// TIA Portal V17 export
// export: Created 2022-07-20T07:02:40.1160452Z, ExportSetting WithDefaults, DisplayName Totally Integrated Automation Portal, DisplayVersion V17, DisplayName TIA Portal Openness, DisplayVersion V17, DisplayName TIA Portal Version Control Interface, DisplayVersion V17, DisplayName SINAMICS Startdrive Advanced, DisplayVersion V17, DisplayName SINAMICS Startdrive G130, G150, S120, S150, SINAMICS MV, S210, DisplayVersion V17, DisplayName SINAMICS Startdrive G110M, G120, G120C, G120D, G120P, G115D, DisplayVersion V17, DisplayName STEP 7 Professional, DisplayVersion V17, DisplayName STEP 7 Safety, DisplayVersion V17, DisplayName WinCC Advanced, DisplayVersion V17
VAR_GLOBAL   // PLC tag table "LAcycCom_Drives"
END_VAR
VAR_GLOBAL CONSTANT   // user constants
   LACYCCOM_WRITE_PARAMETERS_UPPER_LIM : Int := 18;
   LACYCCOM_READ_PARAMETERS_UPPER_LIM : Int := 38;
   LACYCCOM_SILENT_OPERATION_PARAMETERS_UPPER_LIM : Int := 17;
   LACYCCOM_NO_COMMAND : Byte := 16#00;
   LACYCCOM_READ_COMMAND : Byte := 16#01;
   LACYCCOM_WRITE_COMMAND : Byte := 16#02;
   LACYCCOM_TYPE_ALARM : SInt := 1;
   LACYCCOM_TYPE_FAULT : SInt := 2;
   LACYCCOM_TYPE_SI_MESSAGE : SInt := 3;
   LACYCCOM_MESSAGES_UPPER_LIM : Int := 23;
END_VAR
